{attribute 'qualified_only'}
VAR_GLOBAL
END_VAR

(* stored: Version 1.1.0.1, ProductVersion 3.1.4024.16
   GVL GVL: Id {ad778394-f0c0-4082-93ce-56c34f3852fd} *)
